KUKA KRL data list: $robcor.dat

&ACCESS RV
&PARAM VERSION = 1.0.0
&REL 2
DEFDAT $ROBCOR PUBLIC
CHAR $V_ROBCOR[32]
$V_ROBCOR[]="V42.629.9.2/KUKA9.2"
CHAR $MODEL_NAME[32]
$MODEL_NAME[]="#KR140R3200_2PA"
DECL ADAP_ACC $ADAP_ACC=#STEP2
DECL ADAP_ACC $OPT_MOVE=#STEP2
DECL BOOL $OPT_TIME_PTP=FALSE
DECL BOOL $OPT_FLT_PTP=TRUE
DECL CONTROL_PARAMETER $CONTROL_PARAMETER=#STANDARD
BOOL $PROG_TORQ_MON=TRUE
BOOL $ENERGY_MON=TRUE
BOOL $ENERGY_MODULE_ACTIVE=TRUE
INT $OPT_APPROX=100
DECL EKO_MODE $EKO_MODE=#ON
REAL $DEF_L_M=140
FRAME $DEF_L_CM={X 100,Y 0,Z 300,A 0,B 0,C 0}
DECL INERTIA $DEF_L_J={X 70,Y 70,Z 70}
REAL $DEF_LA3_M=50
FRAME $DEF_LA3_CM={X -50,Y 0,Z -1430,A 0,B 0,C 0}
DECL INERTIA $DEF_LA3_J={X 10,Y 10,Z 10}
REAL $RVM_PARAM[4]; Konfigurationsparameter der Resonanzvermeidungsstrategie
$RVM_PARAM[1]=0.0
$RVM_PARAM[2]=0.0
$RVM_PARAM[3]=0.0
$RVM_PARAM[4]=0.0
REAL $LDAA=0.0; Parameter fuer lastabhaengige Beschleunigungsoptimierung
DECL SCARA_VEL_RED_PARAM $SCARA_VEL_RED={DIST_OFFSET 0.0,PAR_LIN 0.0,PAR_QUAD 0.0}; Geschwindigkeitsreduzierung fuer Scarakinematiken
REAL $EKO_DAT[400]
$EKO_DAT[1]=1
$EKO_DAT[2]=32.0
$EKO_DAT[3]=2.0
$EKO_DAT[4]=0.0
$EKO_DAT[5]=1
$EKO_DAT[6]=0
$EKO_DAT[7]=1
$EKO_DAT[8]=1
$EKO_DAT[9]=1
$EKO_DAT[10]=0.0
$EKO_DAT[11]=0.0
$EKO_DAT[12]=0.0
$EKO_DAT[13]=1
$EKO_DAT[14]=1
$EKO_DAT[15]=1
$EKO_DAT[16]=0
$EKO_DAT[17]=0
$EKO_DAT[18]=0
$EKO_DAT[19]=0.0
$EKO_DAT[20]=0.0
$EKO_DAT[21]=0.0
$EKO_DAT[22]=0.0
$EKO_DAT[23]=0.0
$EKO_DAT[24]=0.0
$EKO_DAT[25]=26.7891903
$EKO_DAT[26]=40.5702782
$EKO_DAT[27]=29.9497147
$EKO_DAT[28]=0
$EKO_DAT[29]=0
$EKO_DAT[30]=0
$EKO_DAT[31]=0.0
$EKO_DAT[32]=0.0
$EKO_DAT[33]=0.0
$EKO_DAT[34]=0.0
$EKO_DAT[35]=0.0
$EKO_DAT[36]=0.0
$EKO_DAT[37]=48.2542
$EKO_DAT[38]=68.5440445
$EKO_DAT[39]=65.0812073
$EKO_DAT[40]=0
$EKO_DAT[41]=0
$EKO_DAT[42]=0
$EKO_DAT[43]=0.0
$EKO_DAT[44]=0.0
$EKO_DAT[45]=0.0
$EKO_DAT[46]=0.0
$EKO_DAT[47]=0.0
$EKO_DAT[48]=0.0
$EKO_DAT[49]=100
$EKO_DAT[50]=100
$EKO_DAT[51]=100
$EKO_DAT[52]=0
$EKO_DAT[53]=0
$EKO_DAT[54]=0
$EKO_DAT[55]=0.0
$EKO_DAT[56]=0.0
$EKO_DAT[57]=0.0
$EKO_DAT[58]=0.0
$EKO_DAT[59]=0.0
$EKO_DAT[60]=0.0
$EKO_DAT[61]=2149244
$EKO_DAT[62]=3700999
$EKO_DAT[63]=2100999
$EKO_DAT[64]=0
$EKO_DAT[65]=0
$EKO_DAT[66]=0
$EKO_DAT[67]=0.0
$EKO_DAT[68]=0.0
$EKO_DAT[69]=0.0
$EKO_DAT[70]=0.0
$EKO_DAT[71]=0.0
$EKO_DAT[72]=0.0
$EKO_DAT[73]=2149245
$EKO_DAT[74]=3701000
$EKO_DAT[75]=2101000
$EKO_DAT[76]=0
$EKO_DAT[77]=0
$EKO_DAT[78]=0
$EKO_DAT[79]=0.0
$EKO_DAT[80]=0.0
$EKO_DAT[81]=0.0
$EKO_DAT[82]=0.0
$EKO_DAT[83]=0.0
$EKO_DAT[84]=0.0
$EKO_DAT[85]=0.00027391
$EKO_DAT[86]=0.00037632
$EKO_DAT[87]=0.00066454
$EKO_DAT[88]=0
$EKO_DAT[89]=0
$EKO_DAT[90]=0
$EKO_DAT[91]=0.0
$EKO_DAT[92]=0.0
$EKO_DAT[93]=0.0
$EKO_DAT[94]=0.0
$EKO_DAT[95]=0.0
$EKO_DAT[96]=0.0
$EKO_DAT[97]=0.00033492
$EKO_DAT[98]=0.00014189
$EKO_DAT[99]=0.00033755
$EKO_DAT[100]=0
$EKO_DAT[101]=0
$EKO_DAT[102]=0
$EKO_DAT[103]=0.0
$EKO_DAT[104]=0.0
$EKO_DAT[105]=0.0
$EKO_DAT[106]=0.0
$EKO_DAT[107]=0.0
$EKO_DAT[108]=0.0
$EKO_DAT[109]=3049
$EKO_DAT[110]=4510
$EKO_DAT[111]=3049
$EKO_DAT[112]=0
$EKO_DAT[113]=0
$EKO_DAT[114]=0
$EKO_DAT[115]=0.0
$EKO_DAT[116]=0.0
$EKO_DAT[117]=0.0
$EKO_DAT[118]=0.0
$EKO_DAT[119]=0.0
$EKO_DAT[120]=0.0
$EKO_DAT[121]=1
$EKO_DAT[122]=1
$EKO_DAT[123]=1
$EKO_DAT[124]=0
$EKO_DAT[125]=0
$EKO_DAT[126]=0
$EKO_DAT[127]=0.0
$EKO_DAT[128]=0.0
$EKO_DAT[129]=0.0
$EKO_DAT[130]=0.0
$EKO_DAT[131]=0.0
$EKO_DAT[132]=0.0
$EKO_DAT[133]=532.915482421203
$EKO_DAT[134]=505.850330394464
$EKO_DAT[135]=434.668363777778
$EKO_DAT[136]=33.635
$EKO_DAT[137]=21.9378992
$EKO_DAT[138]=16.7846064932812
$EKO_DAT[139]=0.0
$EKO_DAT[140]=0.0
$EKO_DAT[141]=0.0
$EKO_DAT[142]=0.0
$EKO_DAT[143]=0.0
$EKO_DAT[144]=0.0
$EKO_DAT[145]=241.102707
$EKO_DAT[146]=365.132477
$EKO_DAT[147]=269.547424
$EKO_DAT[148]=0
$EKO_DAT[149]=0
$EKO_DAT[150]=0
$EKO_DAT[151]=0.0
$EKO_DAT[152]=0.0
$EKO_DAT[153]=0.0
$EKO_DAT[154]=0.0
$EKO_DAT[155]=0.0
$EKO_DAT[156]=0.0
$EKO_DAT[157]=434.287781
$EKO_DAT[158]=616.896362
$EKO_DAT[159]=585.730835
$EKO_DAT[160]=0
$EKO_DAT[161]=0
$EKO_DAT[162]=0
$EKO_DAT[163]=0.0
$EKO_DAT[164]=0.0
$EKO_DAT[165]=0.0
$EKO_DAT[166]=0.0
$EKO_DAT[167]=0.0
$EKO_DAT[168]=0.0
$EKO_DAT[169]=100
$EKO_DAT[170]=100
$EKO_DAT[171]=100
$EKO_DAT[172]=0
$EKO_DAT[173]=0
$EKO_DAT[174]=0
$EKO_DAT[175]=0.0
$EKO_DAT[176]=0.0
$EKO_DAT[177]=0.0
$EKO_DAT[178]=0.0
$EKO_DAT[179]=0.0
$EKO_DAT[180]=0.0
$EKO_DAT[181]=0.0
$EKO_DAT[182]=0.0
$EKO_DAT[183]=0.0
$EKO_DAT[184]=0.0
$EKO_DAT[185]=0.0
$EKO_DAT[186]=0.0
$EKO_DAT[187]=0.0
$EKO_DAT[188]=0.0
$EKO_DAT[189]=0.0
$EKO_DAT[190]=0.0
$EKO_DAT[191]=0.0
$EKO_DAT[192]=0.0
$EKO_DAT[193]=0.0
$EKO_DAT[194]=0.0
$EKO_DAT[195]=0.0
$EKO_DAT[196]=0.0
$EKO_DAT[197]=0.0
$EKO_DAT[198]=0.0
$EKO_DAT[199]=0.0
$EKO_DAT[200]=0.0
$EKO_DAT[201]=0.0
$EKO_DAT[202]=0.0
$EKO_DAT[203]=0.0
$EKO_DAT[204]=0.0
$EKO_DAT[205]=0.0
$EKO_DAT[206]=0.0
$EKO_DAT[207]=0.0
$EKO_DAT[208]=0.0
$EKO_DAT[209]=0.0
$EKO_DAT[210]=0.0
$EKO_DAT[211]=0.0
$EKO_DAT[212]=0.0
$EKO_DAT[213]=0.0
$EKO_DAT[214]=0.0
$EKO_DAT[215]=0.0
$EKO_DAT[216]=0.0
$EKO_DAT[217]=0.0
$EKO_DAT[218]=0.0
$EKO_DAT[219]=0.0
$EKO_DAT[220]=0.0
$EKO_DAT[221]=0.0
$EKO_DAT[222]=0.0
$EKO_DAT[223]=0.0
$EKO_DAT[224]=0.0
$EKO_DAT[225]=0.0
$EKO_DAT[226]=0.0
$EKO_DAT[227]=0.0
$EKO_DAT[228]=0.0
$EKO_DAT[229]=0.0
$EKO_DAT[230]=0.0
$EKO_DAT[231]=0.0
$EKO_DAT[232]=0.0
$EKO_DAT[233]=0.0
$EKO_DAT[234]=0.0
$EKO_DAT[235]=0.0
$EKO_DAT[236]=0.0
$EKO_DAT[237]=0.0
$EKO_DAT[238]=0.0
$EKO_DAT[239]=1
$EKO_DAT[240]=3500000
$EKO_DAT[241]=1.001
$EKO_DAT[242]=0
$EKO_DAT[243]=0
$EKO_DAT[244]=0
$EKO_DAT[245]=0
$EKO_DAT[246]=0
$EKO_DAT[247]=0
$EKO_DAT[248]=0
$EKO_DAT[249]=0
$EKO_DAT[250]=0
$EKO_DAT[251]=0
$EKO_DAT[252]=0
$EKO_DAT[253]=0
$EKO_DAT[254]=0
$EKO_DAT[255]=0
$EKO_DAT[256]=0
$EKO_DAT[257]=0
$EKO_DAT[258]=0.0
$EKO_DAT[259]=0.0
$EKO_DAT[260]=0.0
$EKO_DAT[261]=0.0
$EKO_DAT[262]=0.0
$EKO_DAT[263]=0.0
$EKO_DAT[264]=0.0
$EKO_DAT[265]=0.0
$EKO_DAT[266]=0.0
$EKO_DAT[267]=0.0
$EKO_DAT[268]=0.0
$EKO_DAT[269]=0.0
$EKO_DAT[270]=0.0
$EKO_DAT[271]=0.0
$EKO_DAT[272]=0.0
$EKO_DAT[273]=0.0
$EKO_DAT[274]=0.0
$EKO_DAT[275]=0.0
$EKO_DAT[276]=0.0
$EKO_DAT[277]=0.0
$EKO_DAT[278]=0.0
$EKO_DAT[279]=0.0
$EKO_DAT[280]=0.0
$EKO_DAT[281]=0.0
$EKO_DAT[282]=0.0
$EKO_DAT[283]=0.0
$EKO_DAT[284]=0.0
$EKO_DAT[285]=0.0
$EKO_DAT[286]=0.0
$EKO_DAT[287]=0.0
$EKO_DAT[288]=0.0
$EKO_DAT[289]=0.0
$EKO_DAT[290]=0.0
$EKO_DAT[291]=0.0
$EKO_DAT[292]=0.0
$EKO_DAT[293]=0.0
$EKO_DAT[294]=0.0
$EKO_DAT[295]=0.0
$EKO_DAT[296]=0.0
$EKO_DAT[297]=0.0
$EKO_DAT[298]=0.0
$EKO_DAT[299]=0.0
$EKO_DAT[300]=0.0
$EKO_DAT[301]=0.0
$EKO_DAT[302]=0.0
$EKO_DAT[303]=0.0
$EKO_DAT[304]=0.0
$EKO_DAT[305]=0.0
$EKO_DAT[306]=0.0
$EKO_DAT[307]=0.0
$EKO_DAT[308]=0.0
$EKO_DAT[309]=0.0
$EKO_DAT[310]=0.0
$EKO_DAT[311]=0.0
$EKO_DAT[312]=0.0
$EKO_DAT[313]=0.0
$EKO_DAT[314]=0.0
$EKO_DAT[315]=0.0
$EKO_DAT[316]=0.0
$EKO_DAT[317]=0.0
$EKO_DAT[318]=0.0
$EKO_DAT[319]=0.0
$EKO_DAT[320]=0.0
$EKO_DAT[321]=0.0
$EKO_DAT[322]=0.0
$EKO_DAT[323]=0.0
$EKO_DAT[324]=0.0
$EKO_DAT[325]=0.0
$EKO_DAT[326]=0.0
$EKO_DAT[327]=0.0
$EKO_DAT[328]=0.0
$EKO_DAT[329]=0.0
$EKO_DAT[330]=0.0
$EKO_DAT[331]=0.0
$EKO_DAT[332]=0.0
$EKO_DAT[333]=0.0
$EKO_DAT[334]=0.0
$EKO_DAT[335]=0.0
$EKO_DAT[336]=0.0
$EKO_DAT[337]=0.0
$EKO_DAT[338]=0.0
$EKO_DAT[339]=0.0
$EKO_DAT[340]=0.0
$EKO_DAT[341]=0.0
$EKO_DAT[342]=0.0
$EKO_DAT[343]=0.0
$EKO_DAT[344]=0.0
$EKO_DAT[345]=0.0
$EKO_DAT[346]=0.0
$EKO_DAT[347]=0.0
$EKO_DAT[348]=0.0
$EKO_DAT[349]=0.0
$EKO_DAT[350]=0.0
$EKO_DAT[351]=0.0
$EKO_DAT[352]=0.0
$EKO_DAT[353]=0.0
$EKO_DAT[354]=0.0
$EKO_DAT[355]=0.0
$EKO_DAT[356]=0.0
$EKO_DAT[357]=0.0
$EKO_DAT[358]=0.0
$EKO_DAT[359]=0.0
$EKO_DAT[360]=0.0
$EKO_DAT[361]=0.0
$EKO_DAT[362]=0.0
$EKO_DAT[363]=0.0
$EKO_DAT[364]=0.0
$EKO_DAT[365]=0.0
$EKO_DAT[366]=0.0
$EKO_DAT[367]=0.0
$EKO_DAT[368]=0.0
$EKO_DAT[369]=0.0
$EKO_DAT[370]=0.0
$EKO_DAT[371]=0.0
$EKO_DAT[372]=0.0
$EKO_DAT[373]=0.0
$EKO_DAT[374]=0.0
$EKO_DAT[375]=0.0
$EKO_DAT[376]=0.0
$EKO_DAT[377]=0.0
$EKO_DAT[378]=0.0
$EKO_DAT[379]=0.0
$EKO_DAT[380]=0.0
$EKO_DAT[381]=0.0
$EKO_DAT[382]=0.0
$EKO_DAT[383]=0.0
$EKO_DAT[384]=0.0
$EKO_DAT[385]=0.0
$EKO_DAT[386]=0.0
$EKO_DAT[387]=0.0
$EKO_DAT[388]=0.0
$EKO_DAT[389]=0.0
$EKO_DAT[390]=0.0
$EKO_DAT[391]=0.0
$EKO_DAT[392]=0.0
$EKO_DAT[393]=0.0
$EKO_DAT[394]=0.0
$EKO_DAT[395]=0.0
$EKO_DAT[396]=0.0
$EKO_DAT[397]=0.0
$EKO_DAT[398]=0.0
$EKO_DAT[399]=0.0
$EKO_DAT[400]=0.0
BOOL $EMSTOP_ADAP=TRUE
DECL SPO_REACTION $SPO_REACTION=#MODEL_RAMP_STOP
BOOL $USE_CUSTOM_MODEL=FALSE
CHAR $CUSTOM_MODEL_NAME[32]
$CUSTOM_MODEL_NAME[]=" "
CHAR $CUSTOM_MODEL_VERSION[32]
$CUSTOM_MODEL_VERSION[]=" "
ENDDAT
